// TIA Portal V16 export
// export: Created 2021-08-30T10:49:37.4343076Z, ExportSetting WithDefaults, DisplayName Totally Integrated Automation Portal, DisplayVersion V16 Update 3, DisplayName TIA Portal Version Control Interface, DisplayVersion V16 Update 2, DisplayName TIA Portal Openness, DisplayVersion V16 Update 3, DisplayName TIA Portal Teamcenter Gateway, DisplayVersion V16, DisplayName STEP 7 Professional, DisplayVersion V16 Update 3, DisplayName STEP 7 Safety, DisplayVersion V16, DisplayName WinCC Advanced, DisplayVersion V16 Update 3
TYPE "ET_HW_DI"
// stored: IsFailsafeCompliant false
   STRUCT
      HW_DI : Array[0.."ET_DI"] of Bool;
   END_STRUCT;
END_TYPE
